// TIA Portal V20 export
VAR_GLOBAL   // PLC tag table "Unit1Em7_Servo"
   "BA030AZSBK21.00" AT %I1080.0 : Bool;   // SEPA CLAMP&CUTTER X-AXIS LIMIT SENSOR(-)
   "BA030AZSBK21.01" AT %I1080.1 : Bool;   // SEPA CLAMP&CUTTER X-AXIS HOME SENSOR
   "BA030AZSBK21.02" AT %I1080.2 : Bool;   // SEPA CLAMP&CUTTER X-AXIS LIMIT SENSOR(+)
   "BA030AZSBK21.04" AT %I1080.4 : Bool;   // SEPA GRIPPER X-AXIS LIMIT SENSOR(-)
   "BA030AZSBK21.05" AT %I1080.5 : Bool;   // SEPA GRIPPER X-AXIS HOME SENSOR
   "BA030AZSBK21.06" AT %I1080.6 : Bool;   // SEPA GRIPPER X-AXIS LIMIT SENSOR(+)
   "BA030AZSBK22.05" AT %I1084.5 : Bool;   // SEPA GRIPPER C-AXIS LIMIT SENSOR(+)
   "BA030AZSBK22.06" AT %I1084.6 : Bool;   // SEPA GRIPPER Z-AXIS LIMIT SENSOR(-)
   "BA030AZSBK22.07" AT %I1084.7 : Bool;   // SEPA GRIPPER Z-AXIS LIMIT SENSOR(+)
   "BA030AZSBK22.16" AT %I1085.6 : Bool;   // SEPA GRIPPER Z-AXIS HOME SENSOR
   "BA030AZSBK23.00" AT %I1088.0 : Bool;   // SEPA CLAMP&CUTTER Z-AXIS LIMIT SENSOR(-)
   "BA030AZSBK23.01" AT %I1088.1 : Bool;   // SEPA CLAMP&CUTTER Z-AXIS LIMIT SENSOR(+)
   "BA030AZSBK23.10" AT %I1089.0 : Bool;   // CLAMP&CUTTER Z-AXIS HOME SENSOR
   "BA030AZSBK25.00" AT %I1096.0 : Bool;   // JR WINDER REAR Y-AXIS LIMIT SENSOR(-)
   "BA030AZSBK25.01" AT %I1096.1 : Bool;   // JR WINDER REAR Y-AXIS HOME SENSOR
   "BA030AZSBK25.02" AT %I1096.2 : Bool;   // JR WINDER REAR Y-AXIS LIMIT SENSOR(+)
   "BA030AZSBK25.04" AT %I1096.4 : Bool;   // JR WINDER FRONT Y-AXIS LIMIT SENSOR(-)
   "BA030AZSBK25.05" AT %I1096.5 : Bool;   // JR WINDER FRONT Y-AXIS HOME SENSOR
   "BA030AZSBK26.00" AT %I1100.0 : Bool;   // JR WINDER B-AXIS HOME SENSOR
   "BA030AZSBK25.06" AT %I1096.6 : Bool;   // JR WINDER FRONT Y-AXIS LIMIT SENSOR(+)
   "BA030AZSBK22.04" AT %I1084.4 : Bool;   // SEPA GRIPPER C-AXIS LIMIT SENSOR(-)
   "BA030AZSBK22.14" AT %I1085.4 : Bool;   // SEPA GRIPPER C-AXIS HOME SENSOR
   "BA030AZSBK28.00" AT %I1108.0 : Bool;   // PUSHER ROLLER Z-AXIS LIMIT SENSOR(-)
   "BA030AZSBK28.01" AT %I1108.1 : Bool;   // PUSHER ROLLER Z-AXIS HOME SENSOR
   "BA030AZSBK28.06" AT %I1108.6 : Bool;   // PUSHER ROLLER Z-AXIS LIMIT SENSOR(+)
END_VAR
